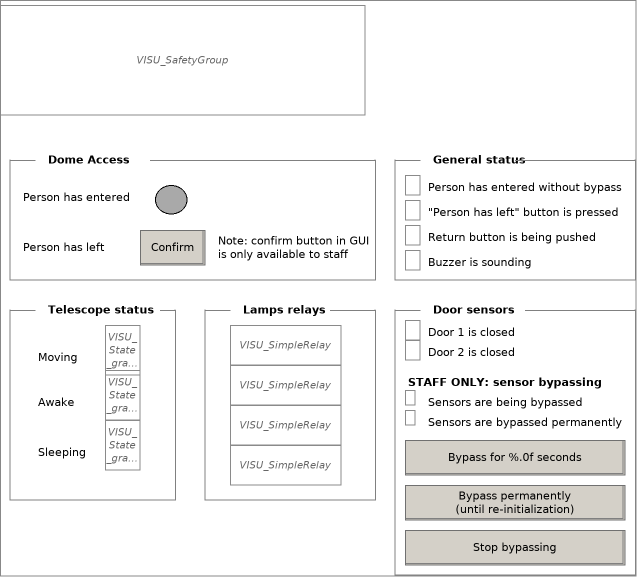
VISUALIZATION VISU_SafetyDomeAccess  // 637x577
VAR_IN_OUT
    ref : SafetyDomeAccess;
    widget : SafetyDomeAccessWidget;
END_VAR
    Polyline (525,310) (635,310) (635,575) (395,575) (395,310) (420,310)
    Polyline (150,160) (375,160) (375,280) (10,280) (10,160) (35,160)
    Label (20,180 130x35), "Person has entered"
    Label (45,150 160x20), "Dome Access"
    Button (140,230 65x35), "Confirm", input disabled if: ref.processes.personHasLeft.statuses.enabledStatus.disabled
        OnMouseClick: execute { ref.processes.personHasLeft.do_request := TRUE; }
    Label (425,395 210x15), "Sensors are being bypassed"
    Button (405,485 220x35), "Bypass permanently (until re-initialization)", input disabled if: ref.processes.bypassPermanently.statuses.enabledStatus.disabled
        OnMouseClick: execute { ref.processes.bypassPermanently.do_request := TRUE; }
    Frame (405,390 10x15)
        shows VISU_State_gray_orange(state := ref.sensorsBeingBypassed)
    Polyline (160,310) (175,310) (175,500) (10,500) (10,310) (35,310)
    Label (45,300 160x20), "Telescope status"
    Label (35,340 65x35), "Moving"
    Frame (105,325 35x50)
        shows VISU_State_gray_red(state := ref.movingLedOn)
    Frame (105,370 35x50)
        shows VISU_State_gray_orange(state := ref.awakeLedOn)
    Label (35,385 60x35), "Awake"
    Frame (105,420 35x50)
        shows VISU_State_gray_green(state := ref.sleepingLedOn)
    Label (35,435 70x35), "Sleeping"
    Label (430,150 105x20), "General status"
    Polyline (515,160) (635,160) (635,280) (395,280) (395,160) (420,160)
    Label (425,325 135x15), "Door 1 is closed"
    Frame (405,320 15x20)
        shows VISU_State_gray_green(state := ref.door1Closed)
    Label (425,345 135x15), "Door 2 is closed"
    Frame (405,340 15x20)
        shows VISU_State_gray_green(state := ref.door2Closed)
    Frame (405,200 15x20)
        shows VISU_State_gray_green(state := ref.personHasLeftButtonPressed)
    Label (425,205 205x15), ""Person has left" button is pressed"
    Frame (405,250 15x20)
        shows VISU_State_gray_yellow(state := ref.buzzerSounding)
    Label (425,255 140x15), "Buzzer is sounding"
    Label (430,300 95x20), "Door sensors"
    Polyline (330,310) (375,310) (375,500) (205,500) (205,310) (230,310)
    Label (240,300 105x20), "Lamps relays"
    Label (215,230 160x35), "Note: confirm button in GUI is only available to staff"
    Label (425,415 210x15), "Sensors are bypassed permanently"
    Frame (405,410 10x15)
        shows VISU_State_gray_orange(state := ref.sensorsBypassedPermanently)
    Label (405,375 210x15), "STAFF ONLY: sensor bypassing"
    Button (405,440 220x35), "Bypass for %.0f seconds", text variable: widget.bypassTimeAfterPassword, input disabled if: ref.processes.bypass.statuses.enabledStatus.disabled
        OnMouseClick: execute { ref.processes.bypass.do_request := TRUE; }
    Button (405,530 220x35), "Stop bypassing", input disabled if: ref.processes.stopBypassing.statuses.enabledStatus.disabled
        OnMouseClick: execute { ref.processes.stopBypassing.do_request := TRUE; }
    Frame (405,175 15x20)
        shows VISU_State_gray_green(state := ref.personHasEntered)
    Label (425,180 210x15), "Person has entered without bypass"
    Frame (230,325 111x40)
        shows VISU_SimpleRelay(ref := ref.parts.lampsRelay1, widget := widget.lampsRelay1)
    Frame (230,365 111x40)
        shows VISU_SimpleRelay(ref := ref.parts.lampsRelay2, widget := widget.lampsRelay2)
    Frame (230,405 111x40)
        shows VISU_SimpleRelay(ref := ref.parts.lampsRelay3, widget := widget.lampsRelay3)
    Frame (230,445 111x40)
        shows VISU_SimpleRelay(ref := ref.parts.lampsRelay4, widget := widget.lampsRelay4)
    Frame (405,225 15x20)
        shows VISU_State_gray_green(state := ref.returnButtonPressed)
    Label (425,230 180x15), "Return button is being pushed"
    Label (20,230 130x35), "Person has left"
    Frame (0,5 365x110)
        shows VISU_SafetyGroup(statusWidget := widget.actualStatus, comError := ref.groupComError, fbError := ref.groupFbError, outError := ref.groupOutError, reset := ref.processes.reset)
    Ellipse (155,185 32x29), colour toggle: ref.personHasEntered
END_VISUALIZATION

(* stored: Version 1.1.0.1, ProductVersion 3.1.4019.2
   Visu VISU_SafetyDomeAccess: Id {066f2eb1-0ae1-468a-a8f7-3ecf9fbfa4ee} *)
